ABB RobotStudio station: Escenario RobotStudio Entregable Práctica 2.rspag

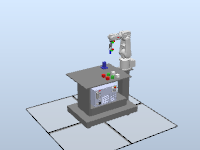
--- station ---
Station Practica2_1920 (saved by RobotStudio 7.0.8732.594)
Controller Controlador_IRC5, task T_ROB1: task frame (RAPID world) sits at (560, 0, 840) mm, rotated rx 0 ry 0 rz 180 deg in the station
Controller Controlador_IRC5
  mechanical unit ROB_1: IRB120_3_58__01, 6 joints, base frame (0, 0, 0) mm
Layout (positions relative to the parent item):
  - Pinza_schunk_SGB50 [mechanism, from Libraries\Pinza_schunk_SGB50.rslib] at (258, 0, 1398) mm, rotated rx 180 ry 0 rz 0 deg; joint values [0, 0.1745, -0.1745] (rad or m)
  - Mesa del robot [part]
  - Cubo XYZ 50 mm 2 [part] at (124, -162, 840) mm, rotated rx 0 ry 0 rz 45 deg
  - Cubo XYZ 50 mm 3 [part] at (200, -150, 840) mm
  - Cubo XYZ 50 mm 4 [part] at (0, -225, 840) mm, rotated rx 0 ry 0 rz -90 deg
  - Cubo XYZ 50 mm 5 [part] at (124, -287, 840) mm, rotated rx 0 ry 0 rz 45 deg
  - Cubo XYZ 50 mm 6 [part] at (200, -275, 840) mm
  - Cubo XYZ 50 mm 1 [part] at (0, -100, 839.71) mm, rotated rx 0 ry 0 rz -90 deg
  - Soporte para elevar los cubos  [part] at (200, 150, 840) mm
  - IRC5_Compact [part, from Equipment\IRC5_Compact__02.rslib] at (-200, -200, 350) mm
  - Soporte para el controlador [part]
  - IRB120_3_58__01 [mechanism, from Robots\IRB120_3_58_G_01.rslib] at (560, 0, 840) mm, rotated rx 0 ry 0 rz 180 deg; joint values [0, 0, 0, 0, 1.5708, 0] (rad or m)
Attachment: Cubo XYZ 50 mm 2 is attached to Mesa del robot
Attachment: Cubo XYZ 50 mm 3 is attached to Mesa del robot
Attachment: Cubo XYZ 50 mm 4 is attached to Mesa del robot
Attachment: Cubo XYZ 50 mm 5 is attached to Mesa del robot
Attachment: Cubo XYZ 50 mm 6 is attached to Mesa del robot
Attachment: Soporte para el controlador is attached to Mesa del robot
Attachment: Pinza_schunk_SGB50 is attached to IRB120_3_58__01 / Link6
EventTableEntry 2988: Group=, Trigger=D16_O 2989, Actions=[EventTableActionMechanicalPose 2990, EventTableActionAttach 2991], Comment=, ActivationMode=2, Cyclic=false
EventTableTriggerIO 2989: IOValue=[1], IRC5Controller=? -1, Operator=0, SignalSource=Controlador_IRC5 2505
EventTableActionMechanicalPose 2990: VirtualSignal=, Mechanism=Pinza_schunk_SGB50 1474, ToPoseName=HomePosition, VirtualSignalValue=[1]
EventTableActionAttach 2991: AttachmentParent=Pinza_schunk_SGB50 1474, AttachmentChild=? -1, MountObject=false, Offset=[X=1, Y=0, Z=0, W=0, X=0, Y=1, Z=0, W=0, X=0, Y=0, Z=1, W=0, X=0, Y=0, Z=0, W=1], FlangeIndext=0, FindNearest=true
EventTableEntry 2992: Group=, Trigger=D16_O 2993, Actions=[EventTableActionMechanicalPose 2994, EventTableActionDetach 2995], Comment=, ActivationMode=2, Cyclic=false
EventTableTriggerIO 2993: IOValue=[0], IRC5Controller=? -1, Operator=0, SignalSource=Controlador_IRC5 2505
EventTableActionMechanicalPose 2994: VirtualSignal=, Mechanism=Pinza_schunk_SGB50 1474, ToPoseName=Abierto, VirtualSignalValue=[1]
EventTableActionDetach 2995: AttachmentParent=Pinza_schunk_SGB50 1474, AttachmentChild=? -1

--- Backups/Controlador_IRC5/RAPID/TASK1/PROGMOD/CalibData.mod ---
MODULE CalibData
	PERS tooldata Pinza_schunk_SGB50_1:=[TRUE,[[-16,0,146.4],[1,0,0,0]],[0.1393,[-13.76,0,75.83],[1,0,0,0],0,0,0]];
ENDMODULE

--- Backups/Controlador_IRC5/RAPID/TASK1/PROGMOD/Module1.mod ---
MODULE Module1
    !***********************************************************
    !
    ! Módulo:  Module1
    !
    ! Descripción:
    !   <Introduzca la descripción aquí>
    !
    ! Autor: Diego
    !
    ! Versión: 1.0
    !
    !***********************************************************


    !***********************************************************
    !
    ! Procedimiento Main
    !
    !   Este es el punto de entrada de su programa
    !
    !***********************************************************
    PROC main()
        !Añada aquí su código
    ENDPROC
ENDMODULE

--- Backups/Controlador_IRC5/SYSPAR/EIO.cfg ---
EIO:CFG_1.0:6:1::
#
EIO_SIGNAL:

      -Name "D16_O" -SignalType "DO" -Access "All"
